(* CoDeSys 2.3.9.37 project: Cap11_16.pro *)
(* Libraries: Standard.lib 4.10.05 12:14:46, IecSfc.lib 13.4.06 16:51:28 *)

(* Global variable list: Global_Variables *)
VAR_GLOBAL

   (* Entradas *)
   P : BOOL;
   FCA:BOOL;
  FCC: BOOL;

   (* Salidas *)
   Abrir: BOOL;
   Cerrar : BOOL;

END_VAR

(* POU PLC_PRG, ST *)
PROGRAM PLC_PRG
VAR
END_VAR
Animacion();
Grafcet();
END_PROGRAM

(* POU Animacion, ST *)
PROGRAM Animacion
VAR
    Pos : INT;
END_VAR
IF (Abrir AND Pos>-160) THEN
   Pos:=Pos-3;
END_IF

IF (Cerrar AND POS<0) THEN
   Pos:=Pos+3;
END_IF

FCC:= (Pos>=0) ;
FCA:=(Pos<=-160);
END_PROGRAM

(* POU Grafcet, SFC *)
PROGRAM Grafcet
VAR
END_VAR
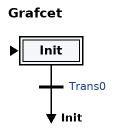
INITIAL_STEP Init:
END_STEP
TRANSITION FROM Init TO Init := Trans0;
END_TRANSITION
END_PROGRAM

(* Visualisation Visu
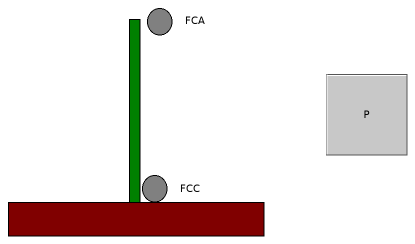
button at (450,140)-(531,221): text "P"; taps P
rectangle at (253,85)-(264,269): bottom Animacion.Pos
ellipse at (266,241)-(291,268): alarm colour if FCC
ellipse at (271,74)-(296,101): alarm colour if FCA
rectangle at (286,244)-(342,265): text "FCC"
rectangle at (291,76)-(347,97): text "FCA"
1 more shapes without text or variables
*)
